TYPE T_LongString : STRING(Param_Configurations.LongStringSize); END_TYPE

(* stored: Version 1.1.0.1, ProductVersion 3.1.4024.4
   DUT T_LongString: Id {d57fe306-93a2-4aa3-9c36-026c7f90ffdc} *)
